// TwinCAT 3 PLC project Untitled1
// ProgramVersion: 3.1.4026.19
// CompilerDefines: VISU_USEPROPERTYINFO
// libraries:
//   Tc2_Standard, * (Beckhoff Automation GmbH)
//   Tc2_System, * (Beckhoff Automation GmbH)
//   VisuSymbols, 4.5.0.0 (System)
// project tree:
//   DUTs/tyCommon/Cylinders/5_3/ ty_Cylinder_5_3_Inputs.TcDUT, ty_Cylinder_5_3_Outputs.TcDUT
//   DUTs/tyCommon/ModeControl/ tyConveyorModeControl.TcDUT
//   DUTs/tyCommon/Motors/ ty_Motor_Inputs.TcDUT, ty_Motor_Outputs.TcDUT
//   / GlobalTextList.TcGTLO, PlcTask.TcTTO, Visualization Manager.TcVMO (not stored)
//   GVLs/ Hmi_Data_Exchange.TcGVL
//   POUs/FbCommon/Cylinders/ Fb_CylinderDualAction_5_3.TcPOU
//   POUs/FbCommon/Motors/ Fb_Motor_Contactor.TcPOU
//   POUs/ MAIN.TcPOU
//   POUs/Project/ fb_BottleTester_Main.TcPOU
//   VISUs/ Visualization.TcVIS

CONFIGURATION Untitled1
    RESOURCE PLC ON TwinCAT3
        TASK PlcTask(INTERVAL := T#10ms, PRIORITY := 20);
        PROGRAM MAIN WITH PlcTask : MAIN;
    END_RESOURCE
END_CONFIGURATION

// ---- DUTs/tyCommon/Cylinders/5_3/ty_Cylinder_5_3_Inputs.TcDUT
TYPE ty_Cylinder_5_3_Inputs :
STRUCT
    bTestMode                    : BOOL;
    bManualMode                  : BOOL;
    
    // Command (Auto)
    b_Reqest_CylinderOut         : BOOL; 
    b_Reqest_CylinderIn          : BOOL; 
    
    // HMI (Manual)
    bHmi_Manual_Reqest_Out       : BOOL; 
    bHmi_Manual_Reqest_In        : BOOL; 
    
    // Physical Feedback Sensors
    bS_Feedback_Sensor_IsOut     : BOOL;
    bS_Feedback_Sensor_IsIn      : BOOL;
    
    // Settings (префикс t_ для типа TIME)
    t_FeedbackSensorDelay        : TIME := T#300MS; 
END_STRUCT
END_TYPE

// ---- DUTs/tyCommon/Cylinders/5_3/ty_Cylinder_5_3_Outputs.TcDUT
TYPE ty_Cylinder_5_3_Outputs :
STRUCT
    // Valve physical outputs
    b_ExtendValve                : BOOL;
    b_RetractValve               : BOOL;
    
    // Feedback status flags
    b_Cylinder_IsExtend            : BOOL;
    b_Cylinder_IsRetract             : BOOL;
    b_ValveError                 : BOOL;
END_STRUCT
END_TYPE

// ---- DUTs/tyCommon/ModeControl/tyConveyorModeControl.TcDUT
{attribute 'qualified_only'}
{attribute 'strict'}
{attribute 'to_string'}
TYPE tyConveyorModeControl :
(
Standby 					:=0,
init 						:=10,
Stopped  					:=20,

//Cycle Steps 
WaitForBottle  				:=30,
OpenInfeedStopper  			:=40,
MoveToTestStation  			:=50,
ExtendTestHead  			:=60,
InjectAir  					:=70,
StabilizeAndMeasure  		:=80,
ReleaseTestHead  			:=90,
ReleaseBottle  				:=100,
RejectBottle  				:=110,

Fault  						:=999
);
END_TYPE

// ---- DUTs/tyCommon/Motors/ty_Motor_Inputs.TcDUT
TYPE ty_Motor_Inputs :
STRUCT
    bTestMode                        : BOOL;
    bManualMode                      : BOOL;
    
    // Command (Auto)
    b_Reqest_SwitchOnMotor           : BOOL;
    
    // HMI (Manual)
    bHmi_Manual_MotorSwitchReqest    : BOOL;
    
    // Physical Feedback (Блок-контакт контактора)
    bS_Feedback_MotorIsRunning       : BOOL;
    
    // Settings
    t_FeedbackDelay                  : TIME := T#300MS;
END_STRUCT
END_TYPE

// ---- DUTs/tyCommon/Motors/ty_Motor_Outputs.TcDUT
TYPE ty_Motor_Outputs :
STRUCT
    // Physical Output (Выход на реле/контактор)
    b_Activate_Contactor             : BOOL;
    
    // Status Flags
    b_Motor_IsRunning                : BOOL;
    b_MotorError                     : BOOL;
END_STRUCT
END_TYPE

// ---- GVLs/Hmi_Data_Exchange.TcGVL
{attribute 'qualified_only'}
VAR_GLOBAL
// -----------------------------------------------------------------------------
//	1. System & Test Mode
// -----------------------------------------------------------------------------	
bTestMode 						:BOOL;
// -----------------------------------------------------------------------------
//	2.Hmi Commands (Buttons)
// -----------------------------------------------------------------------------
bHmiControlOn 					:BOOL;
bHmiControlOFF 					:BOOL;

// -----------------------------------------------------------------------------
//	3. Visu Sensors & Inputs 
// -----------------------------------------------------------------------------
bInfeedCylinderProductVisible	:BOOL;
bTesterProductVisible 		  	:BOOL;
bKickerProductVisible 		  	:BOOL;
bBottleQualityOk	 		  	:BOOL;

// -----------------------------------------------------------------------------
//	4. Machine State
// -----------------------------------------------------------------------------
eCurrentStep : tyConveyorModeControl:= tyConveyorModeControl.Standby;

// -----------------------------------------------------------------------------
//5. Cylinders & Actuators Feedback (Outputs)
// -----------------------------------------------------------------------------
bInfeedCylinderExtend  : BOOL; 
bInfeedCylinderRetract : BOOL; 

bTesterStopperCylinderExtend  : BOOL; 
bTesterStopperCylinderRetract : BOOL; 

bTesterHeadCylinderExtend  : BOOL; 
bTesterHeadCylinderRetract : BOOL; 

bKickerCylinderExtend  : BOOL; 
bKickerCylinderRetract : BOOL; 

bConveyorIsRunning 		:BOOL; 
bAirTestPressureValve 	:BOOL; 

END_VAR

// ---- POUs/MAIN.TcPOU
PROGRAM MAIN
VAR
	BottleTester : fb_BottleTester_Main;
END_VAR

BottleTester ();

END_PROGRAM

// ---- POUs/Project/fb_BottleTester_Main.TcPOU
FUNCTION_BLOCK fb_BottleTester_Main
VAR_INPUT
    bPressureInput_Di                    : BOOL; 
    bCylinder1_ProductOnTheInputStopper  : BOOL;
    bCylinder_ProductOnTheTestStopper    : BOOL;
    bStartPushButton                     : BOOL;
    bStopPushButton                      : BOOL;
    StopperBottleCloseDelay              : TIME := T#2S;
    TestStabilizationTime                : TIME;
    TestBlowTime                         : TIME;
	TesterCylinderExtendTime			 : TIME;
    KickerBottleSensor                   : BOOL;
END_VAR

VAR_OUTPUT
    bPressureValveOut                    : BOOL;

END_VAR

VAR
    eCurrentStep                         : tyConveyorModeControl := tyConveyorModeControl.StandBy;
    eNextStep                            : tyConveyorModeControl := tyConveyorModeControl.StandBy;
    ePrevStep                            : tyConveyorModeControl := tyConveyorModeControl.StandBy;
    
    fbCylinder_InfeedStopper             : Fb_CylinderDualAction_5_3;
    fbCylinder_TestStopper               : Fb_CylinderDualAction_5_3;
    fbCylinder_Kicker                    : Fb_CylinderDualAction_5_3;
    fbCylinder_Tester                    : Fb_CylinderDualAction_5_3;
    fbMotor_Conveyor                     : Fb_Motor_Contactor;
    
    fbStepTimer1                         : TON;
	fbStepTimer2  						: TON;	
    fbBottleKickPulse                    : TP;
    
    bIsRunning                           : BOOL; 
    bKickOutFlag                         : BOOL;
    bStepInit                            : BOOL;
END_VAR

//=============================================================================
// Dmitri Raihtsaum - Copyright 2026
// Created By:     Dmitri Raihtsaum
//-----------------------------------------------------------------------------
// Tested with:    TwinCAT 3
// Engineering:    TwinCAT 3
// Functionality:  BottleTestMachine
// Date:           15.09.2026
// Rev:            0.1
//=============================================================================

// -----------------------------------------------------------------------------
// 1. Input & Hmi paiing  (Read at cycle start )
// -----------------------------------------------------------------------------
bStartPushButton := Hmi_Data_Exchange.bHmiControlOn;
bStopPushButton := Hmi_Data_Exchange.bHmiControlOFF;

bCylinder1_ProductOnTheInputStopper := Hmi_Data_Exchange.bInfeedCylinderProductVisible;
bCylinder_ProductOnTheTestStopper := Hmi_Data_Exchange.bTesterProductVisible;
KickerBottleSensor := Hmi_Data_Exchange.bKickerProductVisible;

// -----------------------------------------------------------------------------
// 2. Control logic (Start/Stop)
// -----------------------------------------------------------------------------
IF bStartPushButton THEN 
	bIsRunning :=TRUE; 	
END_IF

IF bStopPushButton THEN 
	bIsRunning :=FALSE; 	
END_IF

IF NOT bIsRunning THEN 
	eCurrentStep := tyConveyorModeControl.Standby;
	eNextStep 	:= tyConveyorModeControl.Standby;
END_IF

// -----------------------------------------------------------------------------
//3. State Machine 
// -----------------------------------------------------------------------------
CASE eCurrentStep OF 	
// -----------------------------------------------------------------------------
tyConveyorModeControl.Standby: 
// -----------------------------------------------------------------------------

	fbStepTimer1(IN:=FALSE,PT:=T#0MS);
	fbCylinder_InfeedStopper.Extend();
	fbCylinder_Tester.Retract();
	fbCylinder_Kicker.Stop();
	fbCylinder_TestStopper.Stop();
	bPressureValveOut :=FALSE;
	fbMotor_Conveyor.Stop();
	bKickOutFlag :=FALSE;
IF bIsRunning THEN 
eNextStep :=tyConveyorModeControl.WaitForBottle;
END_IF;
// -----------------------------------------------------------------------------
tyConveyorModeControl.WaitForBottle: 
// -----------------------------------------------------------------------------
IF ePrevStep <> eCurrentStep THEN 
fbStepTimer1(IN:=FALSE,PT:=T#0MS);
fbCylinder_InfeedStopper.Extend();
fbCylinder_Tester.Retract();
fbMotor_Conveyor.START();
ELSE
IF bCylinder1_ProductOnTheInputStopper THEN 
	eNextStep :=tyConveyorModeControl.OpenInfeedStopper;
END_IF;
END_IF;

// -----------------------------------------------------------------------------
tyConveyorModeControl.OpenInfeedStopper:
// -----------------------------------------------------------------------------
IF ePrevStep <> eCurrentStep THEN 
fbStepTimer1(IN:=FALSE,PT:=T#0MS);	
fbCylinder_InfeedStopper.Retract();
ELSE 
	fbStepTimer1(IN:=TRUE ,PT:=StopperBottleCloseDelay);
IF fbStepTimer1.Q THEN 
eNextStep :=tyConveyorModeControl.MoveToTestStation;		
END_IF
END_IF
// -----------------------------------------------------------------------------
tyConveyorModeControl.MoveToTestStation: 
// -----------------------------------------------------------------------------
IF ePrevStep <> eCurrentStep THEN 
fbStepTimer1(IN:=FALSE,PT:=T#0MS);
fbCylinder_InfeedStopper.Extend();
fbCylinder_TestStopper.Extend();
fbCylinder_Tester.Retract();
ELSE
	fbStepTimer1(IN:=TRUE ,PT:=T#3S);
IF bCylinder_ProductOnTheTestStopper AND fbStepTimer1.Q THEN 
	eNextStep :=tyConveyorModeControl.ExtendTestHead;	
END_IF
END_IF
// -----------------------------------------------------------------------------
tyConveyorModeControl.ExtendTestHead: 
// -----------------------------------------------------------------------------
IF ePrevStep <> eCurrentStep THEN 
	fbStepTimer1(IN:=FALSE,PT:=T#0MS);
	fbCylinder_Tester.Extend();	

ELSE 
	fbStepTimer1(IN:=TRUE ,PT:=T#3S);
	IF fbCylinder_Tester.CylinderOutput.b_Cylinder_IsExtend AND fbStepTimer1.Q THEN 
		eNextStep :=tyConveyorModeControl.InjectAir;	
	END_IF

END_IF

// -----------------------------------------------------------------------------
tyConveyorModeControl.InjectAir: 
// -----------------------------------------------------------------------------
IF ePrevStep <> eCurrentStep THEN 
	fbStepTimer1(IN:=FALSE,PT:=T#0MS);
	bPressureValveOut :=TRUE; 
	ELSE
		fbStepTimer1(IN:=TRUE ,PT:=T#3S);
		IF fbStepTimer1.Q THEN 
		eNextStep :=tyConveyorModeControl.StabilizeAndMeasure;	
	END_IF
		END_IF

// -----------------------------------------------------------------------------
tyConveyorModeControl.StabilizeAndMeasure: 
// -----------------------------------------------------------------------------
IF ePrevStep <> eCurrentStep THEN 
	fbStepTimer1(IN:=FALSE,PT:=T#0MS);
	bPressureValveOut :=FALSE; 
ELSE 
	fbStepTimer1(IN:=TRUE ,PT:=T#3S);
	IF fbStepTimer1.Q THEN 		
IF NOT bPressureInput_Di THEN 
	bKickOutFlag :=TRUE; 
	END_IF;
	eNextStep :=tyConveyorModeControl.ReleaseTestHead;
	END_IF
END_IF


// -----------------------------------------------------------------------------
tyConveyorModeControl.ReleaseTestHead :
// -----------------------------------------------------------------------------
IF ePrevStep <> eCurrentStep THEN 
	fbStepTimer1(IN:=FALSE,PT:=T#0MS);
	fbCylinder_Tester.Retract();
	ELSE 
		fbStepTimer1(IN:=TRUE ,PT:=T#3S);
	IF fbStepTimer1.Q THEN 	
	eNextStep :=tyConveyorModeControl.ReleaseBottle;
		END_IF;
		END_IF;

// -----------------------------------------------------------------------------
tyConveyorModeControl.ReleaseBottle:
// -----------------------------------------------------------------------------
IF ePrevStep <> eCurrentStep THEN 
fbCylinder_TestStopper.Retract();
fbStepTimer1(IN:=FALSE,PT:=T#0MS);
ELSE
	IF bKickOutFlag THEN 
		eNextStep := tyConveyorModeControl.RejectBottle;
		
		ELSE 
			eNextStep :=tyConveyorModeControl.WaitForBottle;
	END_IF;
	END_IF;
// -----------------------------------------------------------------------------
tyConveyorModeControl.RejectBottle:
// -----------------------------------------------------------------------------
IF ePrevStep <> eCurrentStep THEN
	fbStepTimer1(IN:=FALSE,PT:=T#0MS);
	fbStepTimer2(IN:=FALSE,PT:=T#0MS);
ELSE
	IF KickerBottleSensor THEN 
		fbStepTimer1(IN:=TRUE ,PT:=T#300MS);
		IF fbStepTimer1.Q THEN 
			fbCylinder_Kicker.Extend();
		END_IF
	END_IF
fbStepTimer2(IN:=fbCylinder_Kicker.CylinderOutput.b_Cylinder_IsExtend ,PT:=T#2S);
	IF   fbStepTimer2.q  THEN 
		fbCylinder_Kicker.Retract();
		bKickOutFlag :=FALSE; 
		eNextStep :=tyConveyorModeControl.WaitForBottle;
	END_IF
END_IF;



END_CASE

// -----------------------------------------------------------------------------
// 4. Step Transition
// -----------------------------------------------------------------------------
ePrevStep := eCurrentStep; 
eCurrentStep := eNextStep;


// -----------------------------------------------------------------------------
//5. Hardware & Sub-Block Execution
// -----------------------------------------------------------------------------
//Update simulation mode fefoure FB Call
fbCylinder_InfeedStopper.cylinderInput.bTestMode := Hmi_Data_Exchange.bTestMode;
fbCylinder_TestStopper.cylinderInput.bTestMode := Hmi_Data_Exchange.bTestMode;
fbCylinder_Kicker.cylinderInput.bTestMode:= Hmi_Data_Exchange.bTestMode;
fbCylinder_Tester.cylinderInput.bTestMode:= Hmi_Data_Exchange.bTestMode;
fbMotor_Conveyor.MotorInput.bTestMode := Hmi_Data_Exchange.bTestMode;

//Call Hardware blocks
fbCylinder_InfeedStopper();
fbCylinder_TestStopper();
fbCylinder_Kicker();
fbCylinder_Tester();
fbMotor_Conveyor();

// -----------------------------------------------------------------------------
//6. Output & Hmi Status Mapping
// -----------------------------------------------------------------------------
Hmi_Data_Exchange.eCurrentStep := eCurrentStep;
Hmi_Data_Exchange.bAirTestPressureValve := bPressureValveOut;

//Input mapping from GVL
//bStartPushButton 					:= Hmi_Data_Exchange.bHmiControlOn;
//bStopPushButton  					:= Hmi_Data_Exchange.bHmiControlOFF;
//bCylinder1_ProductOnTheInputStopper := Hmi_Data_Exchange.bInfeedCylinderProductVisible;
//bCylinder_ProductOnTheTestStopper 	:= Hmi_Data_Exchange.bTesterProductVisible;
//KickerBottleSensor 					:= Hmi_Data_Exchange.bKickerProductVisible;
bPressureInput_Di 					:= Hmi_Data_Exchange.bBottleQualityOk;

//Visu /Hmi output mapping
Hmi_Data_Exchange.bInfeedCylinderExtend 		:= fbCylinder_InfeedStopper.CylinderOutput.b_Cylinder_IsExtend;
Hmi_Data_Exchange.bInfeedCylinderRetract 		:= fbCylinder_InfeedStopper.CylinderOutput.b_Cylinder_IsRetract;
Hmi_Data_Exchange.bTesterStopperCylinderExtend	:= fbCylinder_TestStopper.CylinderOutput.b_Cylinder_IsExtend;
Hmi_Data_Exchange.bTesterStopperCylinderRetract := fbCylinder_TestStopper.CylinderOutput.b_Cylinder_IsRetract;
Hmi_Data_Exchange.bTesterHeadCylinderExtend 	:= fbCylinder_Tester.CylinderOutput.b_Cylinder_IsExtend;
Hmi_Data_Exchange.bTesterHeadCylinderRetract 	:= fbCylinder_Tester.CylinderOutput.b_RetractValve;
Hmi_Data_Exchange.bKickerCylinderExtend := fbCylinder_Kicker.CylinderOutput.b_Cylinder_IsExtend;
Hmi_Data_Exchange.bKickerCylinderRetract:= fbCylinder_Kicker.CylinderOutput.b_Cylinder_IsRetract;

Hmi_Data_Exchange.bConveyorIsRunning := fbMotor_Conveyor.MotorOutput.b_Motor_IsRunning;

// -----------------------------------------------------------------------------
// END
// -----------------------------------------------------------------------------

END_FUNCTION_BLOCK

// ---- POUs/FbCommon/Cylinders/Fb_CylinderDualAction_5_3.TcPOU
FUNCTION_BLOCK Fb_CylinderDualAction_5_3
VAR_INPUT
    cylinderInput  : ty_Cylinder_5_3_Inputs;
END_VAR
VAR_OUTPUT
    CylinderOutput : ty_Cylinder_5_3_Outputs ;
END_VAR
VAR
    fbOpenTimer    : TON;
    fbCloseTimer   : TON;
    fbErrorTimer1  : TON;
    fbErrorTimer2  : TON;
END_VAR


// -----------------------------------------------------------------------------
// 1.Solenoid Control (Auto/Man)
// -----------------------------------------------------------------------------
IF NOT cylinderInput.bManualMode THEN 
    CylinderOutput.b_ExtendValve  := cylinderInput.b_Reqest_CylinderOut;
    CylinderOutput.b_RetractValve := cylinderInput.b_Reqest_CylinderIn;
ELSE 
    CylinderOutput.b_ExtendValve  := cylinderInput.bHmi_Manual_Reqest_Out;
    CylinderOutput.b_RetractValve := cylinderInput.bHmi_Manual_Reqest_In;
END_IF;

// -----------------------------------------------------------------------------
// 2. Feedback (Real / Simulation, Testmode)
// -----------------------------------------------------------------------------
IF cylinderInput.bTestMode THEN 
    // Limit Switch simulation
    fbOpenTimer(IN := CylinderOutput.b_ExtendValve AND NOT CylinderOutput.b_RetractValve, PT := cylinderInput.t_FeedbackSensorDelay);
    fbCloseTimer(IN := CylinderOutput.b_RetractValve AND NOT CylinderOutput.b_ExtendValve, PT := cylinderInput.t_FeedbackSensorDelay);
    
    CylinderOutput.b_Cylinder_IsExtend := fbOpenTimer.Q;
    CylinderOutput.b_Cylinder_IsRetract  := fbCloseTimer.Q;
ELSE 
    // Limit switch real sensors read
    CylinderOutput.b_Cylinder_IsExtend := cylinderInput.bS_Feedback_Sensor_IsOut;
    CylinderOutput.b_Cylinder_IsRetract := cylinderInput.bS_Feedback_Sensor_IsIn;
    
    fbOpenTimer(IN := FALSE);
    fbCloseTimer(IN := FALSE);
END_IF;

// -----------------------------------------------------------------------------
// 3. Fault Control 
// -----------------------------------------------------------------------------
fbErrorTimer1(IN := CylinderOutput.b_ExtendValve AND NOT CylinderOutput.b_Cylinder_IsExtend, PT := T#1S);
fbErrorTimer2(IN := CylinderOutput.b_RetractValve AND NOT CylinderOutput.b_Cylinder_IsRetract, PT := T#1S);

CylinderOutput.b_ValveError := fbErrorTimer1.Q OR fbErrorTimer2.Q;

METHOD Extend : BOOL
VAR_INPUT
END_VAR
cylinderInput.b_Reqest_CylinderIn := FALSE;
cylinderInput.b_Reqest_CylinderOut := TRUE;
END_METHOD

METHOD Retract : BOOL
VAR_INPUT
END_VAR
cylinderInput.b_Reqest_CylinderIn := TRUE;
cylinderInput.b_Reqest_CylinderOut := FALSE;
END_METHOD

METHOD Stop : BOOL
VAR_INPUT
END_VAR
cylinderInput.b_Reqest_CylinderIn := FALSE;
cylinderInput.b_Reqest_CylinderOut := FALSE;
END_METHOD

END_FUNCTION_BLOCK

// ---- POUs/FbCommon/Motors/Fb_Motor_Contactor.TcPOU
FUNCTION_BLOCK Fb_Motor_Contactor
VAR_INPUT
    MotorInput     : ty_Motor_Inputs;
END_VAR
VAR_OUTPUT
    MotorOutput    : ty_Motor_Outputs;
END_VAR
VAR
    fbSimTimer     : TON;
    fbErrorTimer1  : TON; // Ошибка: Контактор не включился за 1 сек
    fbErrorTimer2  : TON; // Ошибка: Залипание контактора (обратная связь есть при снятой команде)
END_VAR

// -----------------------------------------------------------------------------
// 1. Contactor Control (Man/Auto)
// -----------------------------------------------------------------------------
IF NOT MotorInput.bManualMode THEN 
    MotorOutput.b_Activate_Contactor := MotorInput.b_Reqest_SwitchOnMotor;
ELSE 
    MotorOutput.b_Activate_Contactor := MotorInput.bHmi_Manual_MotorSwitchReqest;
END_IF;

// -----------------------------------------------------------------------------
// 2. Feedback - contact ( Real + Sim) 
// -----------------------------------------------------------------------------
IF MotorInput.bTestMode THEN 
    // Feedback Emulation
    fbSimTimer(IN := MotorOutput.b_Activate_Contactor, PT := MotorInput.t_FeedbackDelay);
    MotorOutput.b_Motor_IsRunning := fbSimTimer.Q;
ELSE 
    MotorOutput.b_Motor_IsRunning := MotorInput.bS_Feedback_MotorIsRunning;
    fbSimTimer(IN := FALSE);
END_IF;

// -----------------------------------------------------------------------------
// 3. Fault Control
// -----------------------------------------------------------------------------
fbErrorTimer1(IN := MotorOutput.b_Activate_Contactor AND NOT MotorOutput.b_Motor_IsRunning, PT := T#1S);
fbErrorTimer2(IN := NOT MotorOutput.b_Activate_Contactor AND MotorOutput.b_Motor_IsRunning, PT := T#1S);

MotorOutput.b_MotorError := fbErrorTimer1.Q OR fbErrorTimer2.Q;

METHOD Start : BOOL
VAR_INPUT
END_VAR
MotorInput.b_Reqest_SwitchOnMotor :=true;
END_METHOD

METHOD Stop : BOOL
VAR_INPUT
END_VAR
MotorInput.b_Reqest_SwitchOnMotor :=False;
END_METHOD

END_FUNCTION_BLOCK

// ---- GlobalTextList.TcGTLO
TEXTLIST GlobalTextList
  533 = '%s'
  8 = 'OFF'
  664 = 'ON'
  30 = 'Test Mode'
END_TEXTLIST

// ---- VISUs/Visualization.TcVIS
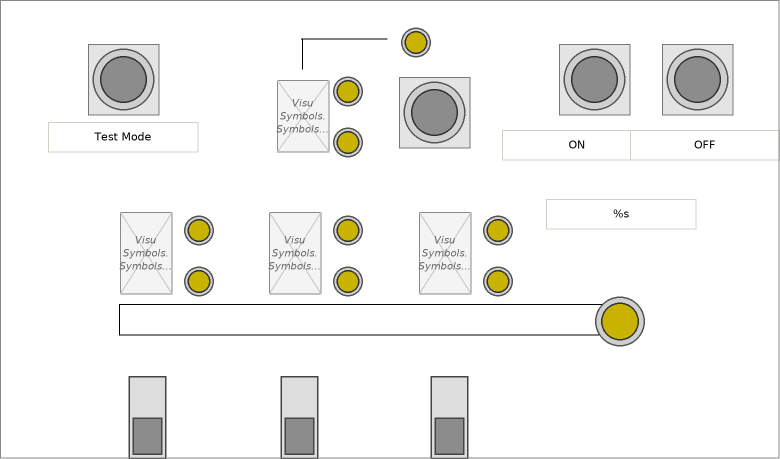
VISUALIZATION Visualization  // 780x459
    Rectangle (119,304 492x31)
    Lamp1 (577,293 86x57), variable: Hmi_Data_Exchange.bConveyorIsRunning, style: Lamp-Lamp1-Yellow
    Lamp1 (182,261 34x41), variable: Hmi_Data_Exchange.bInfeedCylinderRetract, style: Lamp-Lamp1-Yellow
    Lamp1 (182,210 34x41), variable: Hmi_Data_Exchange.bInfeedCylinderExtend, style: Lamp-Lamp1-Yellow
    Lamp1 (331,261 34x41), variable: Hmi_Data_Exchange.bTesterStopperCylinderRetract, style: Lamp-Lamp1-Yellow
    Lamp1 (331,210 34x41), variable: Hmi_Data_Exchange.bTesterStopperCylinderExtend, style: Lamp-Lamp1-Yellow
    Lamp1 (481,261 34x41), variable: Hmi_Data_Exchange.bKickerCylinderRetract, style: Lamp-Lamp1-Yellow
    Lamp1 (481,210 34x41), variable: Hmi_Data_Exchange.bKickerCylinderExtend, style: Lamp-Lamp1-Yellow
    Lamp1 (331,122 34x41), variable: Hmi_Data_Exchange.bTesterHeadCylinderExtend, style: Lamp-Lamp1-Yellow
    Lamp1 (331,71 34x41), variable: Hmi_Data_Exchange.bTesterHeadCylinderRetract, style: Lamp-Lamp1-Yellow
    Image (120,212 52x82), invisible if: NOT Hmi_Data_Exchange.bInfeedCylinderProductVisible, image: VisuSymbols.Symbols.ArrowBoldUp
    Image (269,212 52x82), invisible if: NOT Hmi_Data_Exchange.bTesterProductVisible, image: VisuSymbols.Symbols.ArrowBoldUp
    Image (419,212 52x82), invisible if: NOT Hmi_Data_Exchange.bKickerProductVisible, image: VisuSymbols.Symbols.ArrowBoldUp
    DipSwitch (105,376 85x83), variable: Hmi_Data_Exchange.bInfeedCylinderProductVisible, behaviour: TOGGLE, style: Switch-DipSwitch-Gray
    DipSwitch (257,376 85x83), variable: Hmi_Data_Exchange.bTesterProductVisible, behaviour: TOGGLE, style: Switch-DipSwitch-Gray
    DipSwitch (407,376 85x83), variable: Hmi_Data_Exchange.bKickerProductVisible, behaviour: TOGGLE, style: Switch-DipSwitch-Gray
    PushSwitch (88,40 71x79), variable: Hmi_Data_Exchange.bTestMode, behaviour: TOGGLE, style: Switch-PushSwitch-Gray
    PushSwitch (559,40 71x79), variable: Hmi_Data_Exchange.bHmiControlOn, behaviour: TOGGLE, style: Switch-PushSwitch-Gray
    PushSwitch (662,40 71x79), variable: Hmi_Data_Exchange.bHmiControlOFF, behaviour: TOGGLE, style: Switch-PushSwitch-Gray
    Image (277,80 52x72), image: VisuSymbols.Symbols.ArrowBoldDown
    Lamp1 (399,22 34x41), variable: Hmi_Data_Exchange.bAirTestPressureValve, style: Lamp-Lamp1-Yellow
    Line (387,39) (301,39)
    Line (302,39) (302,69)
    Textfield (502,130 150x30), "ON"
    Textfield (630,130 150x30), "OFF"
    Textfield (48,122 150x30), "Test Mode"
    Textfield (546,199 150x30), "%s", text variable: Hmi_Data_Exchange.eCurrentStep
    PushSwitch (399,73 71x79), variable: Hmi_Data_Exchange.bBottleQualityOk, behaviour: TOGGLE, style: Switch-PushSwitch-Gray
END_VISUALIZATION
